{attribute 'linkalways'} 
{attribute 'no_explicit_call' := 'This FB is a CLASS and must be accessed using methods or properties'}
{attribute 'enable_dynamic_creation'}
FUNCTION_BLOCK CollectionDisposedEvent EXTENDS CollectionEvent IMPLEMENTS I_CollectionDisposedEvent

END_FUNCTION_BLOCK

(* stored: Version 1.1.0.1, ProductVersion 3.1.4024.12
   POU CollectionDisposedEvent: Id {3a0d0f26-5e68-0f29-2e8c-7693d126209c}, SpecialFunc None *)
